// TIA Portal V20 export
FUNCTION_BLOCK "Startup_FB"   // FB9, LAD
{ S7_Optimized_Access := 'TRUE' }
// stored: SetENOAutomatically false
BEGIN

REGION Network 1 (SCL)

   "R_TRIG_DB"(CLK:="FirstScan");
   IF "R_TRIG_DB".Q = 1 THEN
       "GD_Data".Counter_00 := "GD_Data".Counter_00 +1
       ;
   END_IF;
END_REGION
END_FUNCTION_BLOCK
